(* IEC 61131-3 sources: Industry-PLC-LLM/data/PLCBEAD_repo/PLCBEAD_PLCEmbed-main/PLC-BEAD/Source/GEB/DATE_TO_DWORD, 1 file *)

(* ---- DATE_TO_DWORD.ST ---- *)
FUNCTION DATE_TO_DWORD2:DWORD
	VAR_INPUT
		IN :	UDINT;
	END_VAR

	DATE_TO_DWORD2 := UDINT_TO_DWORD(IN);
END_FUNCTION

PROGRAM program0
  VAR
    LocalVar0 : UDINT;
	LocalOUT  : DWORD;
  END_VAR
  	LocalOUT := DATE_TO_DWORD2(LocalVar0);
END_PROGRAM
